FUNCTION_BLOCK AlPgnRxNew8Bcylc (* Receive data cyclic *)
  (* Standard: 61499-2 *)
  (* Version 1.0, 2025-09-04, Franz Höpfinger, initial API and implementation and/or initial documentation *)
  PACKAGE isobus::pgn::rx;
  IMPORT eclipse4diac::core::TypeHash;
  IMPORT isobus::pgn::CAN_MSG;
  IMPORT isobus::pgn::ISONETEVENT_T;
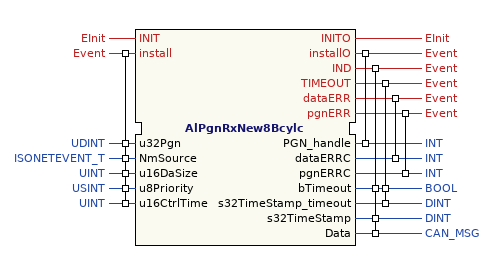
  EVENT_INPUT
    INIT : EInit; (* Service Initialization *)
    install WITH u32Pgn, NmSource, u16DaSize, u8Priority, u16CtrlTime; (* installs a Transmit PGN (TX) *)
  END_EVENT
  EVENT_OUTPUT
    INITO : EInit; (* Initialization Confirm *)
    installO WITH PGN_handle; (* install Done *)
    IND WITH bTimeout, s32TimeStamp, Data; (* Data was received *)
    TIMEOUT WITH bTimeout, s32TimeStamp_timeout;
    dataERR WITH dataERRC;
    pgnERR WITH pgnERRC;
  END_EVENT
  VAR_INPUT
    u32Pgn : UDINT; (* PGN - Range: 0 - 0x3FFFF *)
    NmSource : isobus::pgn::ISONETEVENT_T; (* Define the Communication Partner *)
    u16DaSize : UINT; (* Data length of this PGN (0..8) *)
    u8Priority : USINT := 7; (* Default priority of this PGN (0..7) 0=highest *)
    u16CtrlTime : UINT; (* 0 ... 0xFDFF ms Control time of a receive PGN *)
  END_VAR
  VAR_OUTPUT
    PGN_handle : INT; (* PGN-handle on success, HANDLE_UNVALID in case of an error *)
    dataERRC : INT; (* dataERR error Code *)
    pgnERRC : INT; (* pgnERR error Code *)
    bTimeout : BOOL := FALSE; (* Timeout occured TRUE = Timeout, FALSE = no Timeout *)
    s32TimeStamp_timeout : DINT; (* Time stamp of the Timeout in ms *)
    s32TimeStamp : DINT := -1; (* Time stamp of the message in ms *)
    Data : isobus::pgn::CAN_MSG; (* data buffer *)
  END_VAR
END_FUNCTION_BLOCK
